SYSTEM HMIcontrolHVAC
  (* Version 1.0, 2020-10-18, chong *)
  APPLICATION hvacApp
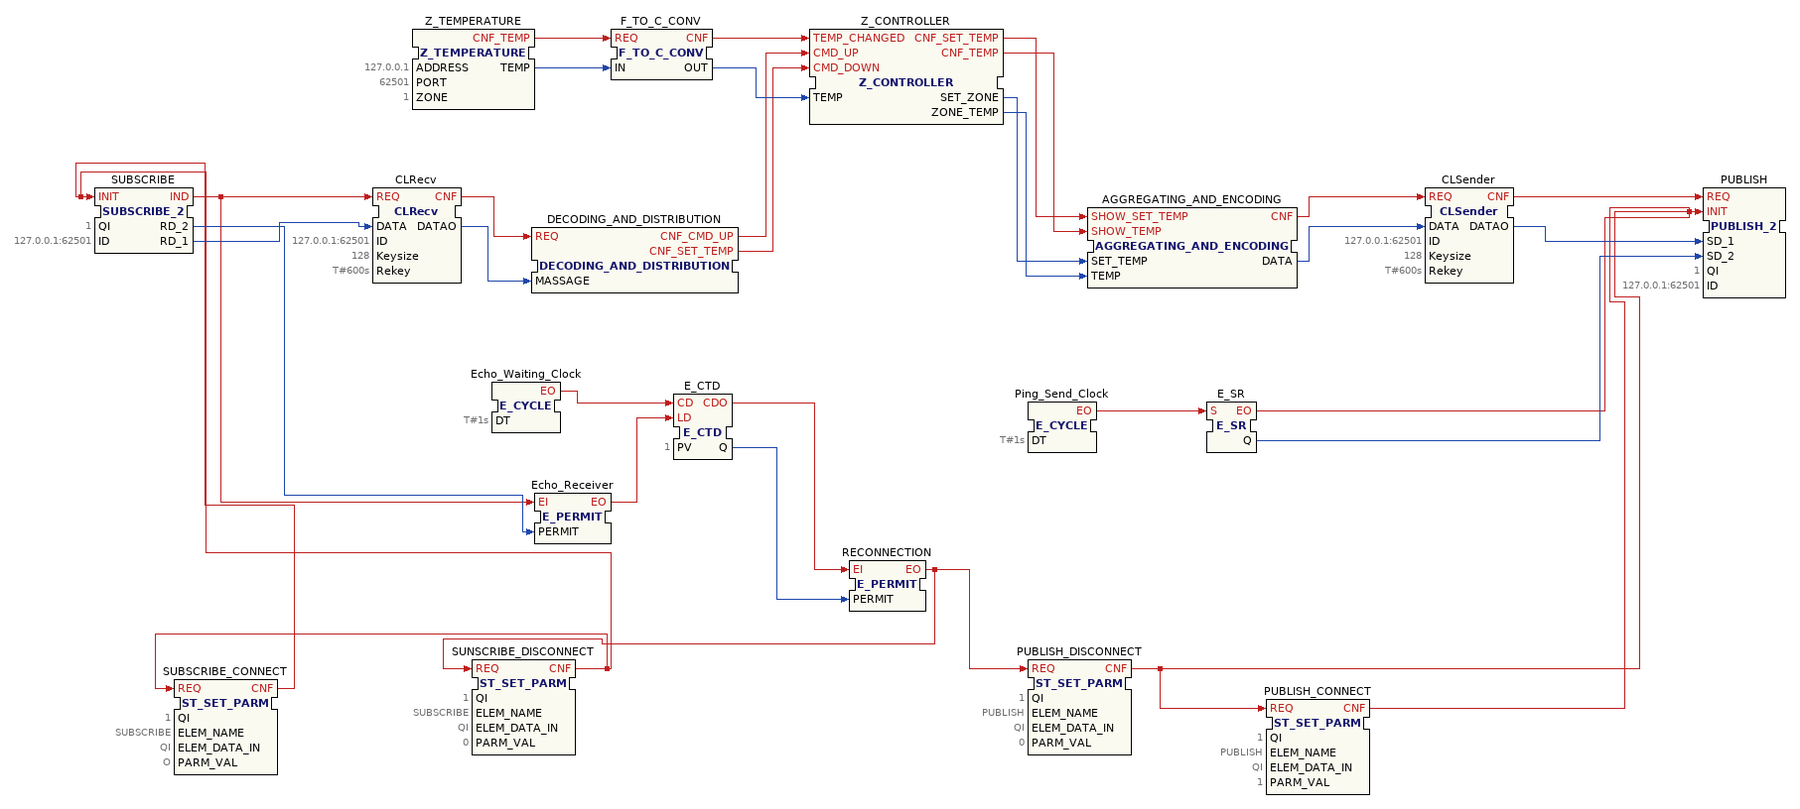
    FBS
      Z_TEMPERATURE : Z_TEMPERATURE(ADDRESS := 127.0.0.1, PORT := 62501, ZONE := 1);
      F_TO_C_CONV : F_TO_C_CONV;
      Z_CONTROLLER : Z_CONTROLLER;
      DECODING_AND_DISTRIBUTION : DECODING_AND_DISTRIBUTION;
      CLRecv : CLRecv(ID := 127.0.0.1:62501, Keysize := 128, Rekey := T#600s);
      AGGREGATING_AND_ENCODING : AGGREGATING_AND_ENCODING;
      CLSender : CLSender(ID := 127.0.0.1:62501, Keysize := 128, Rekey := T#600s);
      Echo_Waiting_Clock : E_CYCLE(DT := T#1s);
      Ping_Send_Clock : E_CYCLE(DT := T#1s);
      E_CTD : E_CTD(PV := 1);
      Echo_Receiver : E_PERMIT;
      RECONNECTION : E_PERMIT;
      PUBLISH : PUBLISH_2(QI := 1, ID := 127.0.0.1:62501);
      SUBSCRIBE : SUBSCRIBE_2(QI := 1, ID := 127.0.0.1:62501);
      PUBLISH_DISCONNECT : ST_SET_PARM(QI := 1, ELEM_NAME := PUBLISH, ELEM_DATA_IN := QI, PARM_VAL := 0);
      PUBLISH_CONNECT : ST_SET_PARM(QI := 1, ELEM_NAME := PUBLISH, ELEM_DATA_IN := QI, PARM_VAL := 1);
      SUNSCRIBE_DISCONNECT : ST_SET_PARM(QI := 1, ELEM_NAME := SUBSCRIBE, ELEM_DATA_IN := QI, PARM_VAL := 0);
      SUBSCRIBE_CONNECT : ST_SET_PARM(QI := 1, ELEM_NAME := SUBSCRIBE, ELEM_DATA_IN := QI, PARM_VAL := O);
      E_SR : E_SR;
    END_FBS
    EVENT_CONNECTIONS
      Z_TEMPERATURE.CNF_TEMP TO F_TO_C_CONV.REQ;
      F_TO_C_CONV.CNF TO Z_CONTROLLER.TEMP_CHANGED;
      DECODING_AND_DISTRIBUTION.CNF_CMD_UP TO Z_CONTROLLER.CMD_UP;
      DECODING_AND_DISTRIBUTION.CNF_SET_TEMP TO Z_CONTROLLER.CMD_DOWN;
      CLRecv.CNF TO DECODING_AND_DISTRIBUTION.REQ;
      Z_CONTROLLER.CNF_SET_TEMP TO AGGREGATING_AND_ENCODING.SHOW_SET_TEMP;
      Z_CONTROLLER.CNF_TEMP TO AGGREGATING_AND_ENCODING.SHOW_TEMP;
      AGGREGATING_AND_ENCODING.CNF TO CLSender.REQ;
      E_CTD.CDO TO RECONNECTION.EI;
      Echo_Waiting_Clock.EO TO E_CTD.CD;
      Echo_Receiver.EO TO E_CTD.LD;
      CLSender.CNF TO PUBLISH.REQ;
      SUBSCRIBE.IND TO Echo_Receiver.EI;
      SUBSCRIBE.IND TO CLRecv.REQ;
      RECONNECTION.EO TO PUBLISH_DISCONNECT.REQ;
      PUBLISH_DISCONNECT.CNF TO PUBLISH.INIT;
      PUBLISH_DISCONNECT.CNF TO PUBLISH_CONNECT.REQ;
      PUBLISH_CONNECT.CNF TO PUBLISH.INIT;
      RECONNECTION.EO TO SUNSCRIBE_DISCONNECT.REQ;
      SUNSCRIBE_DISCONNECT.CNF TO SUBSCRIBE.INIT;
      SUNSCRIBE_DISCONNECT.CNF TO SUBSCRIBE_CONNECT.REQ;
      SUBSCRIBE_CONNECT.CNF TO SUBSCRIBE.INIT;
      Ping_Send_Clock.EO TO E_SR.S;
      E_SR.EO TO PUBLISH.INIT;
    END_CONNECTIONS
    DATA_CONNECTIONS
      Z_TEMPERATURE.TEMP TO F_TO_C_CONV.IN;
      F_TO_C_CONV.OUT TO Z_CONTROLLER.TEMP;
      CLRecv.DATAO TO DECODING_AND_DISTRIBUTION.MASSAGE;
      Z_CONTROLLER.SET_ZONE TO AGGREGATING_AND_ENCODING.SET_TEMP;
      Z_CONTROLLER.ZONE_TEMP TO AGGREGATING_AND_ENCODING.TEMP;
      AGGREGATING_AND_ENCODING.DATA TO CLSender.DATA;
      E_CTD.Q TO RECONNECTION.PERMIT;
      CLSender.DATAO TO PUBLISH.SD_1;
      SUBSCRIBE.RD_2 TO Echo_Receiver.PERMIT;
      SUBSCRIBE.RD_1 TO CLRecv.DATA;
      E_SR.Q TO PUBLISH.SD_2;
    END_CONNECTIONS
  END_APPLICATION
  DEVICE FORTE_PC : FORTE_PC(MGR_ID := "localhost:61499")
    {SET_ATTRIBUTE(Profile, HOLOBLOC)} (* device profile *)
    RESOURCE EMB_RES : EMB_RES
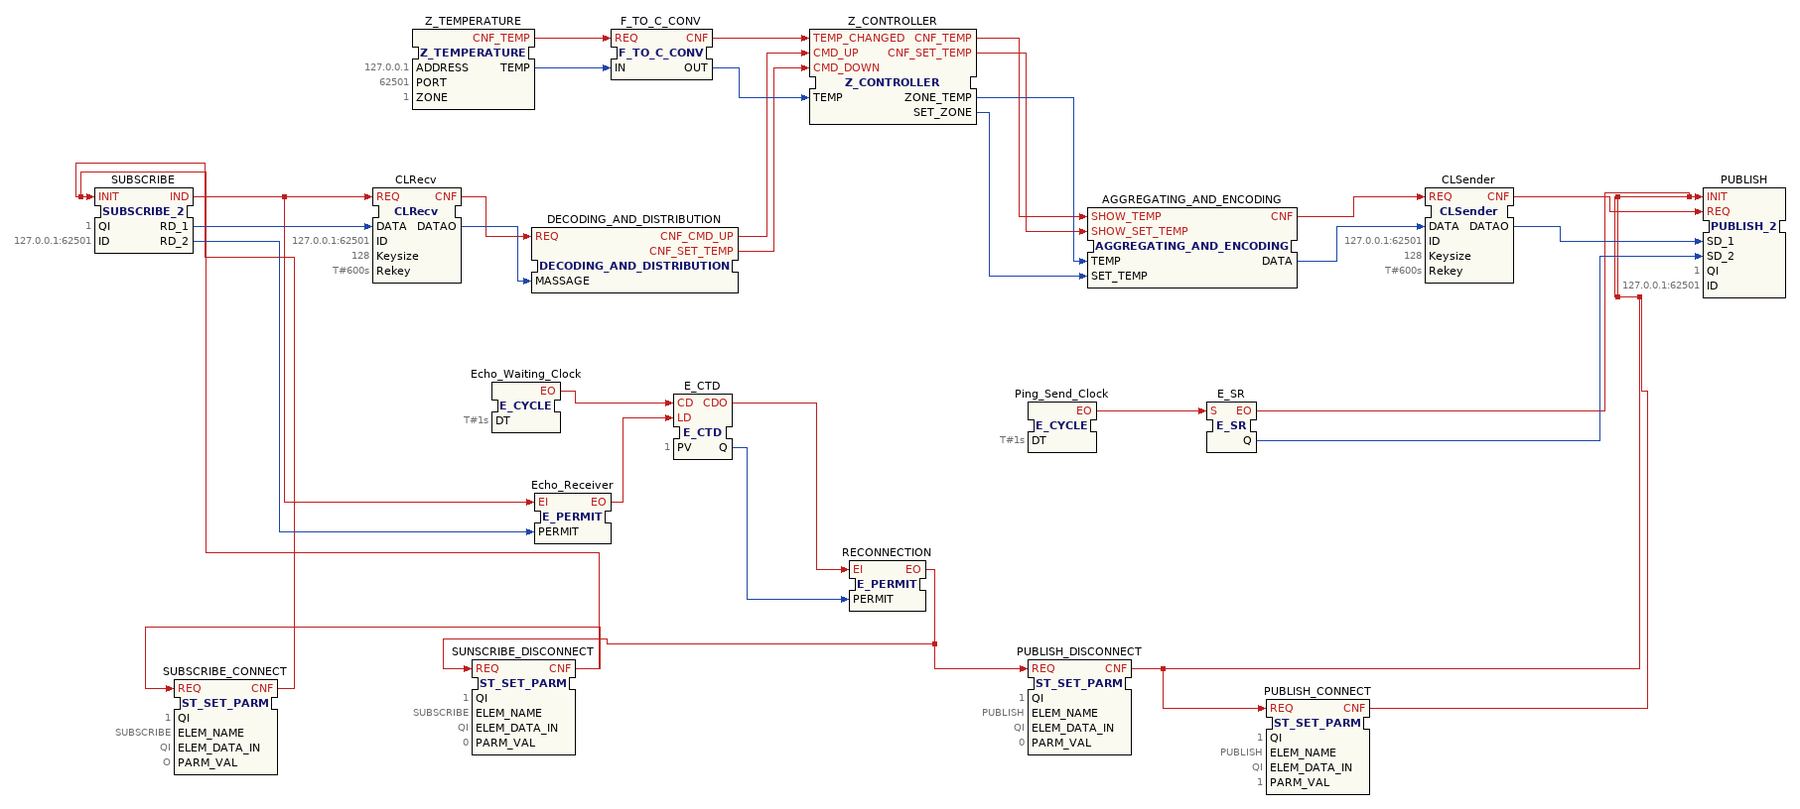
      FBS
        E_CTD : E_CTD(PV := 1);
        Echo_Waiting_Clock : E_CYCLE(DT := T#1s);
        DECODING_AND_DISTRIBUTION : DECODING_AND_DISTRIBUTION;
        PUBLISH_DISCONNECT : ST_SET_PARM(QI := 1, ELEM_NAME := PUBLISH, ELEM_DATA_IN := QI, PARM_VAL := 0);
        F_TO_C_CONV : F_TO_C_CONV;
        AGGREGATING_AND_ENCODING : AGGREGATING_AND_ENCODING;
        Ping_Send_Clock : E_CYCLE(DT := T#1s);
        Z_CONTROLLER : Z_CONTROLLER;
        CLSender : CLSender(ID := 127.0.0.1:62501, Keysize := 128, Rekey := T#600s);
        SUBSCRIBE : SUBSCRIBE_2(QI := 1, ID := 127.0.0.1:62501);
        SUNSCRIBE_DISCONNECT : ST_SET_PARM(QI := 1, ELEM_NAME := SUBSCRIBE, ELEM_DATA_IN := QI, PARM_VAL := 0);
        SUBSCRIBE_CONNECT : ST_SET_PARM(QI := 1, ELEM_NAME := SUBSCRIBE, ELEM_DATA_IN := QI, PARM_VAL := O);
        RECONNECTION : E_PERMIT;
        PUBLISH : PUBLISH_2(QI := 1, ID := 127.0.0.1:62501);
        CLRecv : CLRecv(ID := 127.0.0.1:62501, Keysize := 128, Rekey := T#600s);
        Echo_Receiver : E_PERMIT;
        PUBLISH_CONNECT : ST_SET_PARM(QI := 1, ELEM_NAME := PUBLISH, ELEM_DATA_IN := QI, PARM_VAL := 1);
        Z_TEMPERATURE : Z_TEMPERATURE(ADDRESS := 127.0.0.1, PORT := 62501, ZONE := 1);
        E_SR : E_SR;
      END_FBS
      EVENT_CONNECTIONS
        Echo_Waiting_Clock.EO TO E_CTD.CD;
        F_TO_C_CONV.CNF TO Z_CONTROLLER.TEMP_CHANGED;
        DECODING_AND_DISTRIBUTION.CNF_CMD_UP TO Z_CONTROLLER.CMD_UP;
        DECODING_AND_DISTRIBUTION.CNF_SET_TEMP TO Z_CONTROLLER.CMD_DOWN;
        Z_CONTROLLER.CNF_TEMP TO AGGREGATING_AND_ENCODING.SHOW_TEMP;
        Z_CONTROLLER.CNF_SET_TEMP TO AGGREGATING_AND_ENCODING.SHOW_SET_TEMP;
        AGGREGATING_AND_ENCODING.CNF TO CLSender.REQ;
        SUNSCRIBE_DISCONNECT.CNF TO SUBSCRIBE.INIT;
        SUNSCRIBE_DISCONNECT.CNF TO SUBSCRIBE_CONNECT.REQ;
        SUBSCRIBE_CONNECT.CNF TO SUBSCRIBE.INIT;
        E_CTD.CDO TO RECONNECTION.EI;
        RECONNECTION.EO TO PUBLISH_DISCONNECT.REQ;
        RECONNECTION.EO TO SUNSCRIBE_DISCONNECT.REQ;
        PUBLISH_DISCONNECT.CNF TO PUBLISH.INIT;
        CLSender.CNF TO PUBLISH.REQ;
        SUBSCRIBE.IND TO CLRecv.REQ;
        CLRecv.CNF TO DECODING_AND_DISTRIBUTION.REQ;
        SUBSCRIBE.IND TO Echo_Receiver.EI;
        Echo_Receiver.EO TO E_CTD.LD;
        PUBLISH_DISCONNECT.CNF TO PUBLISH_CONNECT.REQ;
        PUBLISH_CONNECT.CNF TO PUBLISH.INIT;
        Z_TEMPERATURE.CNF_TEMP TO F_TO_C_CONV.REQ;
        Ping_Send_Clock.EO TO E_SR.S;
        E_SR.EO TO PUBLISH.INIT;
      END_CONNECTIONS
      DATA_CONNECTIONS
        F_TO_C_CONV.OUT TO Z_CONTROLLER.TEMP;
        Z_CONTROLLER.ZONE_TEMP TO AGGREGATING_AND_ENCODING.TEMP;
        Z_CONTROLLER.SET_ZONE TO AGGREGATING_AND_ENCODING.SET_TEMP;
        AGGREGATING_AND_ENCODING.DATA TO CLSender.DATA;
        E_CTD.Q TO RECONNECTION.PERMIT;
        CLSender.DATAO TO PUBLISH.SD_1;
        SUBSCRIBE.RD_1 TO CLRecv.DATA;
        CLRecv.DATAO TO DECODING_AND_DISTRIBUTION.MASSAGE;
        SUBSCRIBE.RD_2 TO Echo_Receiver.PERMIT;
        Z_TEMPERATURE.TEMP TO F_TO_C_CONV.IN;
        E_SR.Q TO PUBLISH.SD_2;
      END_CONNECTIONS
    END_RESOURCE
  END_DEVICE
  MAPPINGS
    hvacApp.E_CTD ON FORTE_PC.EMB_RES.E_CTD;
    hvacApp.Echo_Waiting_Clock ON FORTE_PC.EMB_RES.Echo_Waiting_Clock;
    hvacApp.DECODING_AND_DISTRIBUTION ON FORTE_PC.EMB_RES.DECODING_AND_DISTRIBUTION;
    hvacApp.PUBLISH_DISCONNECT ON FORTE_PC.EMB_RES.PUBLISH_DISCONNECT;
    hvacApp.F_TO_C_CONV ON FORTE_PC.EMB_RES.F_TO_C_CONV;
    hvacApp.AGGREGATING_AND_ENCODING ON FORTE_PC.EMB_RES.AGGREGATING_AND_ENCODING;
    hvacApp.Ping_Send_Clock ON FORTE_PC.EMB_RES.Ping_Send_Clock;
    hvacApp.Z_CONTROLLER ON FORTE_PC.EMB_RES.Z_CONTROLLER;
    hvacApp.CLSender ON FORTE_PC.EMB_RES.CLSender;
    hvacApp.SUBSCRIBE ON FORTE_PC.EMB_RES.SUBSCRIBE;
    hvacApp.SUNSCRIBE_DISCONNECT ON FORTE_PC.EMB_RES.SUNSCRIBE_DISCONNECT;
    hvacApp.SUBSCRIBE_CONNECT ON FORTE_PC.EMB_RES.SUBSCRIBE_CONNECT;
    hvacApp.RECONNECTION ON FORTE_PC.EMB_RES.RECONNECTION;
    hvacApp.PUBLISH ON FORTE_PC.EMB_RES.PUBLISH;
    hvacApp.CLRecv ON FORTE_PC.EMB_RES.CLRecv;
    hvacApp.Echo_Receiver ON FORTE_PC.EMB_RES.Echo_Receiver;
    hvacApp.PUBLISH_CONNECT ON FORTE_PC.EMB_RES.PUBLISH_CONNECT;
    hvacApp.Z_TEMPERATURE ON FORTE_PC.EMB_RES.Z_TEMPERATURE;
    hvacApp.E_SR ON FORTE_PC.EMB_RES.E_SR;
  END_MAPPINGS
END_SYSTEM
